{region '#Template'}
	{attribute 'Version' := '1.2.0.0'}
	{attribute 'Tags' := '"LCID": "1031", "Text": "General, Building"'}
	{attribute 'Tags' := '"LCID": "1033", "Text": "General, Building"'}
	{attribute 'Description' := '"LCID": "1031", "Text": "Aufruf Gebäude Funktionen"'}
	{attribute 'Description' := '"LCID": "1033", "Text": "Call building functions"'}
{endregion}
FUNCTION_BLOCK FB_BA_BuildingGlobal EXTENDS FB_BA_View
VAR_INPUT CONSTANT
	BuildAlm			: FB_BA_BuildingAlarms;
	BuildMode			: FB_BA_BuildingMode;
END_VAR

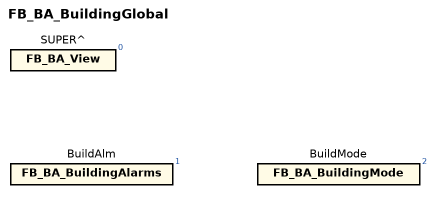
SUPER^(); // FB_BA_View
BuildAlm(); // FB_BA_BuildingAlarms
BuildMode(); // FB_BA_BuildingMode

METHOD FB_init : BOOL
VAR_INPUT
	bInitRetains : BOOL; // if TRUE, the retain variables are initialized (warm start / cold start)
	bInCopyCode : BOOL;  // if TRUE, the instance afterwards gets moved into the copy code (online change)
END_VAR
BuildAlm.iParent			:= THIS^;	
BuildAlm.iLabel				:= LblCmpGeneral.BuildingGlobal_BuildAlm;
BuildAlm.sObjectName		:= '{Idx=01}';											 
BuildAlm.eDPADMode			:= E_BA_DPADMode.eInclude;
                        
BuildMode.iParent			:= THIS^;	
BuildMode.iLabel			:= LblCmpGeneral.BuildingGlobal_BuildMode;
BuildMode.sObjectName		:= '{Idx=02}';											 
BuildMode.eDPADMode			:= E_BA_DPADMode.eInclude;
END_METHOD

END_FUNCTION_BLOCK

(* stored: Version 1.1.0.1, ProductVersion 3.1.4024.9
   POU FB_BA_BuildingGlobal: Id {9830bb13-d0c3-45b7-8e75-802976d1258b}, SpecialFunc None
   Method FB_init: Id {a6f07ee1-7743-4954-833b-5f5fe58694ad} *)
